(* CODESYS project utilitieslib.library
   Author: Chris van Kooij
   Placeholder: Utilities_Library
   Title: Utilities_Library
   Version: 1.2.0.1
   Description: Utilities library contains all basic utilities needed like system variables messages parameters etc.
   Company: AMKO-Engineering

Project tree, tasks and I/O mapping:
  libraries: Tc2_Standard, * (Beckhoff Automation GmbH); Tc2_System, * (Beckhoff Automation GmbH); Tc2_Utilities, * (Beckhoff Automation GmbH)
  Compare/
    Functions/
      function Between [ST]
      function Between360deg [ST]
  Conversion/
    function DegS_To_Rpm [ST]
    function DegS_To_Rpm_And_MMin [ST]
    function Grey_To_Bin [ST]
    function MMin_To_Rpm_And_DegS [ST]
    function Rpm_To_DegS [ST]
  FaultsAndMessages/
    DataTypes/
      data type E_ComponentTypes
      data type E_FaultTypes
      data type E_Locations
      data type E_MessageNumbers
      data type UDT_Fault
    Functions/
      function block Fb_FaultHandler [ST]: CheckEntryValid, ExecCleanUpArray, ExecResetFaults, ExecSetFaultBit, ExecWriteMessage, CmdAddFault
      function block FB_OperatorMessageDisplay [ST]
    global variables Param_Messages
  General/
    DataTypes/
      data type Udt_TimerBandwith
  GVLs/
    global variables DataManager
    global variables GVL_Message
    global variables GVL_Parameters
    global variables GVL_Safety
    global variables Sys_Variables
  Parameter/
    DataTypes/
      Old/
        data type UDT_Parameter_1
        data type Udt_Parameter_2
        data type Udt_ParameterRetain
      data type E_ParameterNames
      data type Udt_Parameter
      data type Udt_ParameterId
      data type Udt_ParLog
    Functions/
      function block FB_ParameterHandler [ST]: CmdAddParameter, ExecChangeParValues
      function block Fb_ParameterHandlerOld [ST]: Mod_SearchIndex, Mod_WriteTeachValue
      function block Fb_ParLogging [ST]: Init, Mod_CSVFileRead, Mod_CSVFileWrite, Mod_BackupPar, Mod_ChangePar, Mod_ReadAllPar
      global variables Param_Settings
  PathFunctions/
    function F_FBNameFromPath [ST]
  Positions/
    FunctionBlocks/
      function block FB_PositionTrigger [ST]: CalcTriggerCompensation, ExecArmTrigger, ExecTurnoverCheck, CmdArmTrigger, CmdSetTriggerPos
    Functions/
      function F_AccDecDistanceFromTime [ST]
      function F_AccDecDistanceFromVelo [ST]
      function F_PosCheck [ST]
      function F_TopVelocityFromTime [ST]
      function F_TriggerPosOffset [ST]
  System/
    DataTypes/
    Functions/
      DataManagement/
        function block FB_PersistentDataManager [ST]: Write
      function block Fb_SystemVariables [ST]
  Utilities_CD
*)

// FaultsAndMessages/DataTypes/E_ComponentTypes
{attribute 'qualified_only'}
{attribute 'strict'}
{attribute 'to_string'}
TYPE E_ComponentTypes :
(
	// No entry
		NA			:= 0,
	// Actuators 
		Cylinder 	:= 10,
		Axis		:= 11,
	// Buttons 
		EstopButton	:= 20,
		EstopBumper	:= 21,	
		Pushbutton 	:= 22,
		Switch		:= 23,
	// I/O
		SafeIO		:= 30,
		Rio_Box		:= 31,
		Rio_Slot	:= 32,
		Encoder		:= 33,
		DiSensor	:= 34,
	// Drive
		ServoDrive 	:= 40,
	// Operation
		HMI			:= 50,
		RemoteOS	:= 51,
		RemoteDB	:= 52,
	// Assemblies
		Assembly 	:= 60,
		SubAssembly	:= 61,
	// functions
		MainProgram		:= 100,
		StepProgram		:= 101,
		FunctionBlock	:= 102 
)UDINT;
END_TYPE

// FaultsAndMessages/DataTypes/E_FaultTypes
{attribute 'qualified_only'}
{attribute 'strict'}
{attribute 'to_string'}
TYPE E_FaultTypes :
(
	NA	:= 0, // Not applicable
	OM 	:= 1, // Operator message
	MC	:= 2, // Missing condition
	CF	:= 3, // Cycle Fault
	FF	:= 4 // Fatal fault
)UDINT;
END_TYPE

// FaultsAndMessages/DataTypes/E_Locations
{attribute 'qualified_only'}
{attribute 'strict'}
TYPE E_Locations :
(
	MainPLC,
	MainPower_230V, 
	MainPower_24V, 
	MainAirSupply,
	MainScreen,
	MainIO,
	RemoteIO
);
END_TYPE

// FaultsAndMessages/DataTypes/E_MessageNumbers
{attribute 'qualified_only'}
{attribute 'strict'}
TYPE E_MessageNumbers :
(
	// no messages
		NA_NoMessage		:= 0, // no message active
	// System faults
		FF_Unknown 			:= 1, // unknown error occured 
		FF_NoCommunication 	:= 2, // no communication detected
		FF_ComunicationFault:= 3, // Communication error detected (does not match expected com)
		FF_Overload			:= 4, // hardware overload detected
		FF_EncoderFault		:= 5, // encoder signal incorrect or not present
		FF_SlaveFault		:= 6, // slave system is has active fatal fault
		FF_AxisFault		:= 7, // Axis fault feedback
		FF_DriveFault		:= 8, // Axis drive fault
		FF_Collision		:= 9, // Collision detected between 2 or more parts of the machine
	// Hardware faults
		CF_FeedbackFault		:= 100,	// Hardware feedback is does not match expected
		CF_WrongDirection		:= 101, // Hardware moving in incorrect direction
		CF_MoveToFast			:= 102, // Hardware movement completion time is lower then minimum
		CF_MoveToSlow			:= 103, // hardware movement maximum time was exceeded
		CF_WrongPosition		:= 104,	// Hardware is at different position then expected
		CF_Obstruction			:= 105, // Obstruction detected in movement path
	// Missing conditions
		MC_WaitingForproduct	:= 200,	// Waiting for product
		MC_WaitingForOperator	:= 201, // Waiting for operator action
		MC_WaitingForModule		:= 202,	// Waiting for other module
		MC_WaitingForMaster		:= 203, // Waiting Waiting for master
		MC_WaitingForSlave		:= 204, // waiting for slave
		MC_WrongPosition		:= 205, // Action or command not possible in current position
	// Operator messages
		OM_AlmostEmpty			:= 300, // product is almost empty refil is required
		OM_Finished 			:= 301, // product or action is finished
		OM_ready				:= 302, // ready for new task
	// Test Messages
		FF_MessageTest			:= 900, // Fatal fault message test
		CF_MessageTest			:= 901, // Cycle fault message test
		MC_MessageTest			:= 902, // Missing condition message test
		OM_MessageTest			:= 903	// Operator message test
)UDINT;
END_TYPE

// FaultsAndMessages/DataTypes/UDT_Fault
TYPE UDT_Fault :
STRUCT
	// active 
		Active 			: BOOL 				:= FALSE;
	// Message type
 		FaultType 		: E_FaultTypes 		:= E_FaultTypes.NA; // Type of message
	// Message Id number used for translation
		MessageNumber 	: UDINT				:= 0; // message number
		LocationNumber	: UDINT 			:= 0; // message number array ([1]= System, [2]= Module,[3]= sub module, [4]= Component)
	// Message discription
		Discription 	: STRING 			:= ''; // Message text discription in english (service personel only)
	// Location
		LocationName	: STRING			:= ''; // Location discription name
		ComponentType 	: E_ComponentTypes 	:= E_ComponentTypes.NA; // Part type discription
	// Time stamp
		StartTime		: DATE_AND_TIME 	:= DT#2020-1-1-00:00:00 ; // Time and date of message occurence
		EndTime			: DATE_AND_TIME		:= DT#2020-1-1-00:00:00 ; // Time and date of message end
	// Module number
		nModuleID		: UDINT 			; // module reference number used for fault, enable, reset, and safety functions (default := 1, 0 = main system)
	// CompleteFaultnumber for visualization
		FullFaultId		: STRING 			:= 'NA.0.0.0'; // Full fault id for use in HMI is writen by fault function [fault type, message#, location#,ComponentType]
END_STRUCT
END_TYPE

// General/DataTypes/Udt_TimerBandwith
TYPE Udt_TimerBandwith :
STRUCT
	Minimal	:LREAL;// Timer values, Minimum time
	Nominal	:LREAL;// timer values, nominal time
	Maximum	:LREAL;// Timer values, Maximum time
END_STRUCT
END_TYPE

// Parameter/DataTypes/Old/UDT_Parameter_1
TYPE UDT_Parameter_1 EXTENDS Udt_ParameterRetain:
STRUCT
	Name		: STRING	; // Parameter data, Parameter name
	Number		: INT		; // Parameter data, Parameter number
	Par_TYPE	: STRING	; // Parameter data, Type of parameter [Mpar, Cpar, Opar, Ppar]
	Discription	: STRING	; // Parameter data, Parmater discription
	Factory		: LREAL		; // Parameter data, Factory standard value
	Maximum		: LREAL		; // Parameter data, Maximum parameter value
	Minimum		: LREAL		; // Parameter data, Minimum parameter value
	Unit		: STRING	; // Parameter data, Unit of measurement
END_STRUCT
END_TYPE

// Parameter/DataTypes/Old/Udt_Parameter_2
TYPE Udt_Parameter_2 :
STRUCT
	bActive		: BOOL 	; // True if parameter is active in machine 
	IndexNumber	: UDINT	; // [Column 0] Array row index number  
	Number		: INT	; // [Column 1]Parameter data, parameter number
	Name		: STRING; // [Column 2]Parameter data, Parameter name
	Par_Type	: STRING; // [Column 3]Parameter data, Type of parameter [Mpar, Cpar, Opar, Ppar]
	Discription	: STRING; // [Column 4]Parameter data, Parmater discription
	Factory		: LREAL	; // [Column 5]Parameter data, Factory standard value
	Maximum		: LREAL	; // [Column 6]Parameter data, Maximum parameter value
	Minimum		: LREAL	; // [Column 7]Parameter data, Minimum parameter value
	Unit		: STRING; // [Column 8]Parameter data, Unit of measurement
	Value		: LREAL	; // [Column 9]Parameter data, Current (active) parameter value
	Saved		: LREAL	; // [Column 10]Parameter data, Saved value or standard setpoint
	bCmdTeach	: BOOL	; // Teach command for devices 
	bCmdSave	: BOOL 	; // Command to parameter handler to save the parameter
//	LastChange	: DT	; // [Column 11]Parameter data, Date of last change
END_STRUCT
END_TYPE

// Parameter/DataTypes/Old/Udt_ParameterRetain
TYPE Udt_ParameterRetain :
STRUCT
	PrepValue	: LREAL		; // Parameter data, prepared value
	Value		: LREAL		; // Parameter data, Current (active) parameter value
	Saved		: LREAL		; // Parameter data, Saved value or standard setpoint
	LastChange	: DT		; // Parameter data, Date of last change
END_STRUCT
END_TYPE

// Parameter/DataTypes/E_ParameterNames
{attribute 'qualified_only'}
{attribute 'strict'}
TYPE E_ParameterNames :
(
	Mpar_StitchLengthLong 			,
	MPar_StitchLengthShort 			,
	MPar_MaxSpeed 					,
	Mpar_MinSpeed 					,
	Mpar_ManualMaxSpeed 			,
	Mpar_BacktackSpeed 				,
	Mpar_SlowEndSpeed 				,
	Mpar_HomingSpeed 				,
	Mpar_CuttingSpeed 				,
	Mpar_MaxAcceleration 			,
	Mpar_MaxDeceleration 			,
	Mpar_Jerk 						,
	Mpar_BacktackAcceleration 		,
	Mpar_BacktackDeceleration 		,
	Mpar_TransferAcceleration 		,
	Mpar_TransferDeceleration 		,
	Mpar_CylinderTimeoutMargin		,
	Cpar_NeedleSensorPos 			,
	Cpar_NeedlePosUp 				,
	Cpar_NeedlePosInMaterial 		,
	Cpar_NeedleposDown 				,
	Cpar_NeedlePosStartCut 			,
	Cpar_NeedlePosStopCut 			,
	Cpar_NeedlePosEndCut 			,
	Cpar_NeedlePosRelTensCut 		,
	Cpar_NeedlePosHoldThread 		,
	Cpar_NeedlePosStartRelTension 	,
	Cpar_NeedlePosStopRelTension 	,
	Cpar_NeedlePosChangeDirUp 		,
	Cpar_NeedlePosClearStart 		,
	Cpar_NeedlePosClearEnd 			,
	Cpar_NeedlePosRef 				,
	Cpar_NeedlePosPause 			,
	Cpar_SensorPreEdgeDetDistance 	,
	Cpar_sensorEdgeDetDistance 		,
	Opar_NeedleSensorPos 			,
	Opar_NeedlePosUp 				,
	Opar_NeedlePosInMaterial 		,
	Opar_NeedleposDown 				,
	Opar_NeedlePosStartCut 			,
	Opar_NeedlePosStopCut 			,
	Opar_NeedlePosEndCut 			,
	Opar_NeedlePosRelTensCut 		,
	Opar_NeedlePosHoldThread 		,
	Opar_NeedlePosStartRelTension 	,
	Opar_NeedlePosStopRelTension 	,
	Opar_NeedlePosChangeDir 		,
	Opar_NeedlePosClearStart 		,
	Opar_NeedlePosClearEnd 			,
	Opar_NeedlePosPause 			,
	Ppar_BacktackStitchStartFwd 	,
	Ppar_BacktackStitchStartRev 	,
	Ppar_BacktackStitchEndFwd 		,
	Ppar_BacktackStitchEndRev 		,
	Ppar_AutomaticSpeed 			,
	Ppar_StitchStretch 				,
	Ppar_ThreadLengthAdition 		,
	Ppar_ThreadBreakDelay 			,
	Mpar_MaxVelocity 				,
	Mpar_MinVelocity 				,
	Mpar_ManualMaxVelocity 			,
	Mpar_MLTMaxAcceleration 		,
	Mpar_MLTMaxDeceleration 		,
	Mpar_TraverseLength 			,
	Mpar_CylTimeOutMargine 			,
	Mpar_HomingVelocity 			,
	Mpar_SewingcartLength 			,
	Mpar_ClampCartLength 			,
	Mpar_MaxClampCartVelocity 		,
	Mpar_TraverseReturnVelocity 	,
	Mpar_ToStartvelocity 			,
	Mpar_InspectionDistance 		,
	Cpar_PosHoming 					,
	Cpar_PosSuportCyl_1 			,
	Cpar_PosSuportCyl_2 			,
	Cpar_PosSuportCyl_3 			,
	Cpar_PosService 				,
	Cpar_PosBobinChange 			,
	Cpar_PosEnd 					,
	Cpar_TimeBaseClampsClose 		,
	Cpar_TimeBaseClampsRel 			,
	Cpar_TimeCartClampsClose 		,
	Cpar_TimeCartClampsRel 			,
	Cpar_TimeCartBrakeApply 		,
	Cpar_TimeCartBrakeRel 			,
	Cpar_TimeSupportExp_1 			,
	Cpar_TimeSupportRet_1 			,
	Cpar_TimeSupportExp_2 			,
	Cpar_TimeSupportRet_2 			,
	Cpar_TimeSupportExp_3 			,
	Cpar_TimeSupportRet_3 			,
	Cpar_TimeBobinPlateClose 		,
	Cpar_TimeBobinPlateOpen 		,
	Cpar_PosFlagSewingcart 			,
	Cpar_PosSensorClampCart 		,
	Cpar_SupportCylWidth 			,
	Cpar_ClampCartFlagWidth 		,
	Cpar_PosMaterialStart 			,
	Opar_HomePosition 				,
	Opar_PosSuportCyl_1 			,
	Opar_PosSuportCyl_2 			,
	Opar_PosSuportCyl_3 			,
	Opar_PosService 				,
	Opar_PosBobinChange 			,
	Opar_PosEnd 					,
	Opar_PosMatStart 				,
	Ppar_ProductLenght 				,
	Ppar_ProductStretch 			,
	Ppar_StartStretchFactor 		,
	Ppar_StartStretchLength 		,
	Ppar_ReverseStretch 			,
	Ppar_MatBlowDistance 			 
)UDINT;
END_TYPE

// Parameter/DataTypes/Udt_Parameter
TYPE Udt_Parameter :
STRUCT
	nNumber		: INT	 	:= 0				; // [Column 1]Parameter data, parameter number
	sName		: STRING	:= 'No parameter' 	; // [Column 2]Parameter data, Parameter name
	sType		: STRING	:= 'PPar'			; // [Column 3]Parameter data, Type of parameter [Mpar, Cpar, Opar, Ppar]
	sDiscription: STRING	:= 'No parameter selcted'; // [Column 4]Parameter data, Parmater discription
	fFactory	: LREAL		:= 0				; // [Column 5]Parameter data, Factory standard value
	fMaximum	: LREAL		:= 0				; // [Column 6]Parameter data, Maximum parameter value
	fMinimum	: LREAL		:= 0				; // [Column 7]Parameter data, Minimum parameter value
	sUnit		: STRING	:= 'na'				; // [Column 8]Parameter data, Unit of measurement
	fValue		: LREAL		:= 0				; // [Column 9]Parameter data, Current (active) parameter value
	fSaved		: LREAL		:= 0				; // Parameter data, Saved value or standard setpoint
	fPrepared	: LREAL 	:= 0				; // Parameter data, Prepared value from teach function 
	bCmdTeach	: BOOL		:= FALSE			; // Teach command for devices 
END_STRUCT
END_TYPE

// Parameter/DataTypes/Udt_ParameterId
TYPE Udt_ParameterId :
STRUCT
	nNumber		: INT 		:= 0 	; // parameter number
	sName		: STRING 	:= 'NA' ; // parameter name
	sType		: STRING 	:= 'Ppar'	; // parameter type 
	pParameter	: POINTER TO Udt_Parameter ; // pointer to parameter
END_STRUCT
END_TYPE

// Parameter/DataTypes/Udt_ParLog
TYPE Udt_ParLog :
STRUCT
	ParList		: ARRAY [0..Param_Settings.MAX_PARAMETERS] OF Udt_Parameter_2 ; // active parameter list
END_STRUCT
END_TYPE

// FaultsAndMessages/Param_Messages
{attribute 'qualified_only'}
VAR_GLOBAL CONSTANT
	nMAX_MESSAGES_SHOWN 	: UDINT := 10 	;
	nMAX_MESSAGE_HISTORY	: UDINT := 1000 ;
	nMAX_CSV_FIELD_LENGTH	: UDINT := 100	;
	tMESSAGE_TIMEOUT		: TIME 	:= T#5S ;
	sLOGFILE_PATH			: STRING:= 'C:\FaultLogs\'	;
	sLOGFILE_NAME			: STRING:= 'Faultlog' 		; // Message log destination file
	nMESSAGE_COLUMNS		: UDINT := 8 ;
	
END_VAR

// GVLs/DataManager
{attribute 'qualified_only'}
VAR_GLOBAL
	FbPersistentManager : FB_PersistentDataManager ;
END_VAR

// GVLs/GVL_Message
{attribute 'qualified_only'}
VAR_GLOBAL
	bResetFaults		: BOOL 	:= FALSE	; // Reset system faults 
	bCmdSnoozeMessage	: BOOL 	:= FALSE	; // Snooze message display
	bDisplayFaults		: BOOL := FALSE 	; // Display fault message popup on screen (when MC, CF of FF are active)
	arActiveFaults 		: ARRAY [0..Param_Messages.nMAX_MESSAGES_SHOWN] OF UDT_Fault ; // Active faults overview for showing in HMI
END_VAR
VAR_GLOBAL CONSTANT 
	tMESSAGESNOOZEDURATION	: TIME 	:= T#5s ; // duration of message snooze after button press 
END_VAR

// GVLs/GVL_Parameters
{attribute 'qualified_only'}
VAR_GLOBAL
	fbParameterHandler	: FB_ParameterHandler ; // Default parameter handler for visualisation and file handling
END_VAR

// GVLs/GVL_Safety
{attribute 'qualified_only'}
VAR_GLOBAL
	// ===== system Safety inputs =====
		SafeCom_SystemSafe		AT %I* : BOOL ; // System safety communication safety system is running
		SafeCom_EstopOk			AT %I* : BOOL ; // System safety communication emergency stop active
		SafeCom_BumpersOk		AT %I* : BOOL ; // System safety communication safety zone tripped
		SafeCom_ComError		AT %I* : BOOL ; // System safety communication Common error active in safety program
		
		SafeCom_EstopReset		AT %Q* : BOOL ; // System Safety Communication Safety Reset 
		SafeCom_RunSafety		AT %Q* : BOOL ; // System Safety Communication Run safety program
		SafeCom_AcnSafeError	AT %Q* : BOOL ; // System Safety Communication acknowlidge safety error		 
		SafeCom_ResetActive		AT %Q* : BOOL ; // System safety communication reset active
		Safecom_BumperReset		AT %Q* : BOOL ; // System safety communication reset safety bumpers 
		SafeCom_EnableOff		AT %Q* : BOOL ; // System Safety communication motor enable signals are off
		
		SafeOp_AirPressureOk	AT %I* : BOOL ; // system safety condition monitorring air pressure ok
		SafeOp_PowerSupplyOk	AT %I* : BOOL ; // System power supply is ok
END_VAR

// GVLs/Sys_Variables
(* System variables *)
{attribute 'qualified_only'}
VAR_GLOBAL
// SystemFuntion
	fbSystemVariables : Fb_SystemVariables ;
	AlwaysOn		:BOOL 			;// System variable, Always on bit
	AlwaysOff		:BOOL 			;// System variable, Always off bit
	BlinkFast		:BOOL 			;// System variable, Blink fast bit 1sec 
	BlinkSlow		:BOOL 			;// System variable, Blink slow bit 2 sec
	Pulse1Sec		:BOOL 			;// System variable, Pulse 1 cycle every second
	SystemTime		:DT				; // System variable, Windows system time
	TimeZoneId		:E_TimeZoneID 	; // System variable, time zone Id 
	HeartBeat		:BOOL 			;// System Variable, Main system heartbeat 0.5 sec on 0.5 sec off
END_VAR

// Parameter/Functions/Param_Settings
{attribute 'qualified_only'}
VAR_GLOBAL CONSTANT
	MAX_PARAMETERS 			: UDINT := 1000	;
	PAR_COLUMNS 			: UDINT := 11	;
	MAX_CSV_FIELD_LENGTH	: UDINT := 100	;
	sPARLIST_FILE			: T_MaxString 		:= 'C:\Users\chris\Documents\TestCsvList.csv';(* CSV destination file path and name *)
	sPARLOG_FILE			: T_MaxString 		:= 'C:\Users\chris\Documents\TestCsvLog.csv';(* CSV destination file path and name *)
	sNetId					: T_AmsNetID		:= '' ;
END_VAR

// Compare/Functions/Between
FUNCTION Between : BOOL // Returns true if value is >= the lower and <= the upper threshold
VAR_INPUT
	Lower	: LREAL	; // lower threshold value [LREAL]
	Value	: LREAL	; // test value [LREAL]
	Upper	: LREAL	; // Upper threshold value [LREAL]
END_VAR
VAR
END_VAR

// Check if value is between lower and upper threshold
Between := (Value >= Lower) AND (Value <= Upper);

END_FUNCTION

// Compare/Functions/Between360deg
FUNCTION Between360deg : BOOL // Returns true if value is >= the lower and <= the upper threshold, if lower > upper then upper := Upper +360 deg
VAR_INPUT
	Lower	: LREAL	; // lower threshold value [LREAL]
	Value	: LREAL	; // test value [LREAL]
	Upper	: LREAL	; // Upper threshold value [LREAL]
END_VAR
VAR
END_VAR

IF Lower > Upper THEN  
	Between360deg S= Between( Lower, Value, 360);
	Between360deg S= Between( 0, Value, Upper)	;
ELSE 
	Between360deg S= Between( Lower, Value, Upper)	;
END_IF

END_FUNCTION

// Conversion/DegS_To_Rpm
(* convert degrees per second to rotations per minute *)
FUNCTION DegS_To_Rpm : LREAL
VAR_INPUT
	DegS : LREAL ; // Input degrees per second as long real
END_VAR

// ===== convert degrees per second to Rpm =====
	DegS_To_Rpm := (DegS/360)*60 ;

END_FUNCTION

// Conversion/DegS_To_Rpm_And_MMin
FUNCTION DegS_To_Rpm_And_MMin : BOOL
VAR_INPUT
	DegPerSecond : LREAL ; // Input degrees per second
	StitchLength : LREAL ; // Input stitch length
END_VAR
VAR_OUTPUT
	RevPerMinute	: LREAL ; // Output revolutions per minute
	MetersPerMinute	: LREAL ; // Output meters per minute
END_VAR
VAR
END_VAR

// ===== convert degrees per second to Rpm =====
	RevPerMinute := (DegPerSecond/360)*60 ;
// ===== Convert RPM to MMin =====
	MetersPerMinute := RevPerMinute * StitchLength / 1000 ;

END_FUNCTION

// Conversion/Grey_To_Bin
FUNCTION Grey_To_Bin : INT // convert 4 bit grey code into 8 bit binary code
VAR_INPUT
	GreyBit0 : BOOL := FALSE ;
	GreyBit1 : BOOL := FALSE ;
	GreyBit2 : BOOL := FALSE ;
	GreyBit3 : BOOL := FALSE ;
END_VAR
VAR
	TempInt : INT ; // temporary 
END_VAR

// convert grey code into binary
TempInt.3 	:= GreyBit3 ;
TempInt.2	:= GreyBit3 	XOR GreyBit2 ;
TempInt.1	:= TempInt.2	XOR GreyBit1 ;
TempInt.0	:= TempInt.1	XOR GreyBit0 ;

Grey_To_Bin := TempInt ;

END_FUNCTION

// Conversion/MMin_To_Rpm_And_DegS
(* Convert meters per minute to degrees per second *)
FUNCTION MMin_To_Rpm_And_DegS : BOOL
VAR_INPUT
	MeterPerMinute 	: LREAL ; // Input meters per minute
	StitchLength	: LREAL ; // Input Stitch length
END_VAR
VAR_OUTPUT
	RevPerMinute	: LREAL ; // Output revolutions per minute
	DegPerSecond	: LREAL ; // Output degrees per second
END_VAR
VAR
	MmMin 	: LREAL ; // Millimeters per minute
	RevSec 	: LREAL ; // Millimeters per second
END_VAR

// ===== convert MMin to RPM =====
	RevPerMinute := (MeterPerMinute * 1000) / StitchLength ;
//===== Convert RPM to DegS =====
	DegPerSecond := (RevPerMinute/60)*360 ;

END_FUNCTION

// Conversion/Rpm_To_DegS
(* convert rotations per minute to degrees per second *)
FUNCTION Rpm_To_DegS : LREAL 
VAR_INPUT
	Rpm : LREAL ; // input revolutions per minute
END_VAR

// ===== convert RPM to DegS ====
	Rpm_To_DegS := (Rpm/60)*360 ;

END_FUNCTION

// FaultsAndMessages/Functions/Fb_FaultHandler
FUNCTION_BLOCK Fb_FaultHandler
VAR_INPUT
	bReset 				: BOOL 	:= FALSE	; // reference to fault reset bit
END_VAR
VAR_OUTPUT
	arActiveFaults 	: ARRAY [0..Param_Messages.nMAX_MESSAGES_SHOWN] OF UDT_Fault  ; // reference to active fault array
	nActiveFaults	: UDINT 			; // reference to active fault counter
	bActOM 			: BOOL := FALSE ;
	bActMC 			: BOOL := FALSE ;
	bActCF 			: BOOL := FALSE ;
	bActFF 			: BOOL := FALSE ;
END_VAR
VAR
	// functional variables
	i 					: UDINT ;
	// fault data
	stFaultUdt 			: UDT_Fault ;
	bTimedOut 			: BOOL ; // Message has timed out
	// Message logging
	dToday				: DATE ; 
	nWriteStep			: UDINT := 0 ;
	bWriteError			: BOOL 	; // write to file error occured
	nWriteErroId		: UDINT ; // write error id
	// Write variables
	sActFileName		: STRING ;
	hFile				: UINT	:= 0;(* File handle of the source file *)
	sMessageString		: ARRAY [0..Param_Messages.nMESSAGE_COLUMNS] OF STRING (Param_Settings.MAX_CSV_FIELD_LENGTH); (* temporary parameter buffer to string*)
	sCSVLine			: T_MaxString := '';(* Single CSV text line (row, record), we are using string as record buffer (your are able to see created fields) *)
	sCSVField			: T_MaxString := '';(* Single CSV field value (column, record field) *)

	// Log to file functions
	fbFileOpen		: FB_FileOpen	;(* Opens file *)
	fbFileClose		: FB_FileClose	;(* Closes file *)
	fbFileGets		: FB_FileGets	;(* Reads one record (line) *)
	fbFilePuts		: FB_FilePuts	;(* Writes one record (line) *)
	fbReader		: FB_CSVMemBufferReader;(* Helper function block used to parse CSV data bytes (single record line) *)
	fbWriter		: FB_CSVMemBufferWriter;(* Helper function block used to create CSV data bytes (single record line) *)
END_VAR
VAR PERSISTENT
	dLastFileDate : DATE ;
END_VAR
VAR CONSTANT
	stEmptyMessageUdt : UDT_Fault := (	Active 			:= FALSE,
										FaultType 		:= E_FaultTypes.NA,
										MessageNumber	:= 0,
										LocationNumber	:= 0,
										Discription 	:= '',
										LocationName	:= '',
										ComponentType	:= E_ComponentTypes.NA,
										StartTime		:= DT#2020-1-1-00:00:00,
										EndTime			:= DT#2020-1-1-00:00:00,
										FullFaultId		:= '0'	)  ;
END_VAR

// Check for active faults in list
ExecSetFaultBit(); 
// Check for reset is active 
ExecResetFaults();

METHOD PRIVATE CheckEntryValid : BOOL
VAR
	// functional variables
	i 	: UDINT ;
END_VAR
// ======= check if new entry is valid and not already active ======
CheckEntryValid S= TRUE ;
FOR i := 0 TO nActiveFaults DO
	IF arActiveFaults[i].MessageNumber = stFaultUdt.MessageNumber THEN 
		CheckEntryValid 			:= FALSE ; 
		arActiveFaults[i].Active 	:= TRUE ; 
	END_IF
END_FOR
END_METHOD

METHOD PRIVATE ExecCleanUpArray : BOOL
VAR
	// functional variables
	i 					: UDINT ;
END_VAR
// Clean up array by removing blanc spaces 
REPEAT
	IF arActiveFaults[i].FaultType = 0 THEN 
		arActiveFaults[i] 	:= arActiveFaults[i+1];
		arActiveFaults[i+1] := stEmptyMessageUdt;
	END_IF
	i := i +1 ;
UNTIL 
	i = Param_Messages.nMAX_MESSAGES_SHOWN   
END_REPEAT
END_METHOD

METHOD PRIVATE ExecResetFaults : BOOL
VAR
	nResetPoint : UDINT := 0 ; // point of reset for active fault array (skips fault if .active bit is true)
	// functional variables
	i 					: UDINT ;
END_VAR
IF NOT bReset THEN 
	RETURN;
END_IF

FOR i := 0 TO Param_Messages.nMAX_MESSAGES_SHOWN DO
	IF arActiveFaults[i].Active THEN
		CONTINUE;
	ELSE
		arActiveFaults[i] := stEmptyMessageUdt; 
	END_IF
END_FOR

ExecCleanUpArray();

bActOM 			:= FALSE;
bActMC 			:= FALSE;
bActCF 			:= FALSE;
bActFF 			:= FALSE;

ExecResetFaults := TRUE ;
END_METHOD

METHOD PRIVATE ExecSetFaultBit : BOOL
bActOM 	:= FALSE;
bActMC	:= FALSE;
bActCF 	:= FALSE;
bActFF 	:= FALSE;

FOR i := 0 TO nActiveFaults DO
	// read message type 
	CASE arActiveFaults[i].FaultType OF
		E_FaultTypes.OM : 
			IF arActiveFaults[i].Active THEN 
				bActOM 		S= TRUE ;
			ELSE 
				bTimedOut 	S= TRUE ;
			END_IF 
		E_FaultTypes.MC :
			IF arActiveFaults[i].Active THEN 
				bActMC 		S= TRUE ;
			ELSE 
				bTimedOut 	S= TRUE ;
			END_IF 
		E_FaultTypes.CF:
			bActCF 		S= TRUE ;
		E_FaultTypes.FF:
			bActFF 		S= TRUE ;
		ELSE
			bTimedOut := FALSE ;
	END_CASE

	IF bTimedOut THEN 
		arActiveFaults[i] := stEmptyMessageUdt;				
		bTimedOut := FALSE ;
	END_IF
	// Reset active bit when timed out, if fault is still active it will be set to true again.
	arActiveFaults[i].Active R= (arActiveFaults[i].StartTime + Param_Messages.tMESSAGE_TIMEOUT) < Sys_Variables.SystemTime;
END_FOR

// clean up the fault array
ExecCleanUpArray();
END_METHOD

ACTION ExecWriteMessage:
// Set message start time 
stFaultUdt.StartTime := Sys_Variables.SystemTime ;
// Fill Full Fault Id
stFaultUdt.FullFaultId := TO_STRING(stFaultUdt.FaultType);
stFaultUdt.FullFaultId := CONCAT(stFaultUdt.FullFaultId,'.');
stFaultUdt.FullFaultId := CONCAT(stFaultUdt.FullFaultId,UDINT_TO_STRING(stFaultUdt.MessageNumber));
stFaultUdt.FullFaultId := CONCAT(stFaultUdt.FullFaultId,'.');
stFaultUdt.FullFaultId := CONCAT(stFaultUdt.FullFaultId,UDINT_TO_STRING(stFaultUdt.LocationNumber));
stFaultUdt.FullFaultId := CONCAT(stFaultUdt.FullFaultId,'.');
stFaultUdt.FullFaultId := CONCAT(stFaultUdt.FullFaultId,UDINT_TO_STRING(stFaultUdt.ComponentType));
// send message to higher level 
arActiveFaults[nActiveFaults] := stFaultUdt		;
// Set pointer to next fault
IF nActiveFaults < Param_Messages.nMAX_MESSAGES_SHOWN THEN 
	nActiveFaults := nActiveFaults + 1 	;
ELSE
	nActiveFaults := 0 ;
END_IF
END_ACTION

METHOD PUBLIC CmdAddFault : BOOL
VAR_IN_OUT
	stFault : UDT_Fault ; // actuive fault structure input
END_VAR

// coppy fault to internal fault udt
IF stFault.FaultType <> E_FaultTypes.NA THEN 
	THIS^.stFaultUdt	:= stFault ;
	stFault 			:= stEmptyMessageUdt ;
	stFaultUdt.Active	:= TRUE ;
	// Process fault data
	IF CheckEntryValid() THEN
		ExecWriteMessage();
	END_IF
END_IF
END_METHOD

END_FUNCTION_BLOCK

// FaultsAndMessages/Functions/FB_OperatorMessageDisplay
FUNCTION_BLOCK FB_OperatorMessageDisplay // function compares messages and shows latest message on screen for a set period of time
VAR_INPUT
	bEnable 	: BOOL 	:= TRUE ; // enable messages
	tDisplayTime: TIME	:= Param_Messages.tMESSAGE_TIMEOUT ; // Time before message relevance is checked (default = Param_Messages.tMESSAGE_TIMEOUT)
END_VAR
VAR_IN_OUT
	sMessage 	: STRING ; // Operator message (default = GVL_Message.sOPeratorMessage)
END_VAR
VAR_OUTPUT
	sOutMessage : STRING ; // message output to screen
END_VAR
VAR
	sOldMessage 	: STRING := ''; // old message as displayed 
	tonDisplayTimer	: TON ; // Display timer
END_VAR

// Run timers
tonDisplayTimer(PT := tDisplayTime);

// compare old message with new message 
IF sMessage = sOldMessage THEN 
	tonDisplayTimer.IN := TRUE ;
	IF tonDisplayTimer.Q = TRUE THEN 
		sMessage := '';
	END_IF
ELSE 
	tonDisplayTimer.IN 	:= FALSE 	;
	sOldMessage 		:= sMessage ; 
END_IF

// write message to display
sOutMessage := sMessage ;

END_FUNCTION_BLOCK

// Parameter/Functions/FB_ParameterHandler
FUNCTION_BLOCK PUBLIC FB_ParameterHandler
VAR_INPUT
END_VAR
VAR_OUTPUT
	arParameters		: ARRAY [0..Param_Settings.MAX_PARAMETERS] OF Udt_ParameterId := [stDummyParId]; 
END_VAR
VAR
	nLookupIndex		: UDINT := 0;
	nNumberOfParameters : UDINT := 0;
	// parameter change commands
	bCmdLoadfactory		: BOOL 	:= FALSE; // Load factory value into prepared value 
	bCmdLoadFromPrevious: BOOL 	:= FALSE; // Load from saved previous value into prepared value
	bCmdTeach			: BOOL 	:= FALSE; // Start teaching function for selected parameter
	bCmdAcceptTeach		: BOOL 	:= TRUE ; // Accept the teach value
	// Dummy parameter when no parameters are added yet
	stDummyParId		: Udt_ParameterId ;
	// Memory 
	fValueOld			: LREAL	:= 0 ; // previous value
END_VAR

// call parameter change function 
ExecChangeParValues();

METHOD PUBLIC CmdAddParameter : BOOL
VAR_INPUT
	refParameter : REFERENCE TO Udt_Parameter ; // reference to parameter 
END_VAR
VAR
	i 			: UDINT ;
	j			: UDINT ;
	stTempPar	: Udt_ParameterId ;
	bParFound	: BOOL 	:= FALSE ;
END_VAR
// check if parameter is already added
FOR i := 0 TO Param_Settings.MAX_PARAMETERS DO
	IF arParameters[i].pParameter = 0 THEN 
		nNumberOfParameters := i;
		EXIT ;
	ELSIF arParameters[i].nNumber = refParameter.nNumber THEN
 		RETURN ;
	END_IF
END_FOR
	
// Add parameter to array if not already added
arParameters[nNumberOfParameters].nNumber		:= refParameter.nNumber 	;
arParameters[nNumberOfParameters].sName			:= refParameter.sName	;
arParameters[nNumberOfParameters].sType			:= refParameter.sType	;
arParameters[nNumberOfParameters].pParameter 	:= ADR(refParameter)	;

IF nNumberOfParameters > 1 THEN 
	// (re)sort parameter list
	FOR i := 0 TO nNumberOfParameters BY 1 DO
		FOR j := 0 TO nNumberOfParameters -1 BY 1 DO
			IF (arParameters[j].nNumber > arParameters[j+1].nNumber)THEN
				stTempPar 			:= arParameters[j+1];
				arParameters[j+1]	:= arParameters[j];
				arParameters[j]		:= stTempPar ;
			END_IF
		END_FOR
	END_FOR	
END_IF

// set feedback
CmdAddParameter S= arParameters[nNumberOfParameters].pParameter > 0 ;
END_METHOD

METHOD ExecChangeParValues : BOOL
VAR
END_VAR
IF arParameters[nLookupIndex].pParameter <> 0 THEN 
	;
ELSE
	RETURN; 
END_IF

// Load values from default or saved
IF bCmdLoadfactory THEN 
	arParameters[nLookupIndex].pParameter^.fValue := arParameters[nLookupIndex].pParameter^.fValue ;
ELSIF bCmdLoadFromPrevious THEN
	arParameters[nLookupIndex].pParameter^.fValue := arParameters[nLookupIndex].pParameter^.fSaved ;
ELSIF bCmdAcceptTeach THEN 
	arParameters[nLookupIndex].pParameter^.fValue := arParameters[nLookupIndex].pParameter^.fPrepared ;
END_IF

	// Save current actual value for later restore
IF arParameters[nLookupIndex].pParameter^.fValue <> fValueOld THEN
	arParameters[nLookupIndex].pParameter^.fSaved := fValueOld ;
	fValueOld := arParameters[nLookupIndex].pParameter^.fValue ;
END_IF
END_METHOD

END_FUNCTION_BLOCK

// Parameter/Functions/Fb_ParameterHandlerOld
FUNCTION_BLOCK PUBLIC Fb_ParameterHandlerOld EXTENDS Fb_ParLogging 
VAR_INPUT
	bCmdScrollUp	: BOOL 	:= FALSE; // command to scroll to next parameter
	bCmdScrollDown	: BOOL 	:= FALSE; // command to scroll to previous parameter
	bCmdAccept		: BOOL 	:= FALSE; // Accept parameter and coppy prev value into value
	bCmdSave		: BOOL 	:= FALSE; // save active value into memory 
	bCmdLoad		: BOOL 	:= FALSE; // Load value from memory into prepared value
	bCmdRestore		: BOOL 	:= FALSE; // load Factory value into prepared value
	bCmdRestoreAll	: BOOL 	:= FALSE; // Restore all values to factory default
	bCmdSaveToFile 	: BOOL 	:= FALSE; // Save all parameters to .csv file
END_VAR
VAR_IN_OUT
	PrepValue	: LREAL	:= 0 ; // Parameter data, prepared value
END_VAR
VAR_OUTPUT
	stParToHMI	: Udt_Parameter_2 ; // Parameter that can be shown on HMI 
	bReady		: BOOL 	; // function is ready for new command
	bBussy		: BOOL 	; // Function is bussy
	nProgress	: UDINT ; // Progress for visu [%] 
	bDone		: BOOL 	; // Function is done 
END_VAR
VAR
	CmdIndex	: UDINT ; // Index number of parameter
	
	// ====== functions ======
		rtCmdScrollUp	: R_TRIG; // command to scroll to next parameter
		rtCmdScrollDown	: R_TRIG; // command to scroll to previous parameter
		rtCmdAccept		: R_TRIG; // Accept parameter and coppy prev value into value
		rtCmdSave		: R_TRIG; // save active value into memory 
		rtCmdLoad		: R_TRIG; // Load value from memory into prepared value
		rtCmdRestore	: R_TRIG; // load Factory value into prepared value
		rtCmdSaveToFile : R_TRIG; // Save all parameters to .csv file
		rtCmdTeach		: R_TRIG; // Triger 

	// ====== Teach functions =======
		bCmdTeach		: BOOL 	:= FALSE; // Place teach value in parameter

END_VAR

SUPER^();

// ====== Create rising edges ======
	rtCmdScrollUp	(CLK := bCmdScrollup);
	rtCmdScrollDown	(CLK := bCmdScrollDown);
	rtCmdAccept		(CLK := bCmdAccept);
	rtCmdSave		(CLK := bCmdSave);
	rtCmdLoad		(CLK := bCmdLoad);
	rtCmdRestore	(CLK := bCmdRestore);
	rtCmdSaveToFile	(CLK := bCmdSaveToFile);
	rtCmdTeach		(CLK := bCmdTeach);
	
// call search index 
	IF NOT bCmdTeach THEN 
		Mod_SearchIndex();
	END_IF
	
// ====== Always check if prepared value is within min max range ======
	PrepValue := LIMIT (stParLog.ParList[CmdIndex].Minimum, PrepValue, stParLog.ParList[CmdIndex].Maximum);

// ====== process parameter Prep value ======
	IF rtCmdRestore.Q THEN 
		PrepValue := stParLog.ParList[CmdIndex].Factory ;
	ELSIF rtCmdLoad.Q THEN 
		PrepValue := stParLog.ParList[CmdIndex].Saved	;
	ELSIF rtCmdSave.Q THEN 
		stParLog.ParList[CmdIndex].Saved := stParLog.ParList[CmdIndex].Value ; 
	ELSIF rtCmdAccept.Q THEN 
		stParLog.ParList[CmdIndex].Value := PrepValue ;
	ELSIF rtCmdTeach.Q THEN 
		stParLog.ParList[CmdIndex].Value := PrepValue ;
		bCmdTeach 		:= FALSE ;
		bCmdWriteAllPar := TRUE ;
	END_IF		

// ======= check for missing values and restore to factory ======
	IF stParLog.ParList[CmdIndex].Value = 0 AND stParLog.ParList[CmdIndex].Minimum >0 THEN 
		stParLog.ParList[CmdIndex].Value := PrepValue := stParLog.ParList[CmdIndex].Factory ;
	END_IF

// ======= Restore all values to factory default =======
	IF bCmdRestoreAll THEN 
		FOR CmdIndex := 0 TO Param_Settings.MAX_PARAMETERS BY 1 DO
			IF stParLog.ParList[CmdIndex].bActive THEN  
				stParLog.ParList[CmdIndex].Value := PrepValue := stParLog.ParList[CmdIndex].Factory ;
			END_IF
		END_FOR
	END_IF
	
// ======= save parameters to file =======
	IF rtCmdSaveToFile.Q THEN
		bCmdWriteAllPar := TRUE ;
	END_IF
		 
// ======= set feedback to HMI =====
	stParToHMI :=  stParLog.ParList[CmdIndex] ;
	
	IF bWriteBusy OR bReadBusy THEN 
		bReady		:= FALSE;
		bBussy 		:= TRUE ;
		nProgress 	:= (100 / Param_Settings.MAX_PARAMETERS)* nRow ;
	ELSE
		bReady		:= TRUE	;
		bBussy 		:= FALSE;
		nProgress 	:= (100 / Param_Settings.MAX_PARAMETERS)* nRow ;
	END_IF

METHOD PRIVATE Mod_SearchIndex : BOOL
VAR_INPUT
END_VAR
// ====== set scroll index ======
	IF rtCmdScrollUp.Q THEN 
		 CmdIndex := CmdIndex + 1 ;
	ELSIF rtCmdScrollDown.Q THEN 
		 CmdIndex := CmdIndex - 1 ;
	END_IF 	 
	
// check if index number is within reach and if parameter is active
	IF CmdIndex > Param_Settings.MAX_PARAMETERS THEN 
		CmdIndex := 0 ;
	ELSIF CmdIndex < 0 THEN
		CmdIndex := Param_Settings.MAX_PARAMETERS ;
	END_IF

	IF NOT stParLog.ParList[CmdIndex].bActive AND bCmdScrollUp THEN // go to next index if parameter is not active 
		IF CmdIndex < Param_Settings.MAX_PARAMETERS THEN
			CmdIndex := CmdIndex + 1 ;
		ELSE
			CmdIndex := 0 ;
		END_IF
	ELSIF NOT stParLog.ParList[CmdIndex].bActive AND bCmdScrollDown THEN // go to previous index if parameter is not active 
		IF CmdIndex > 0 THEN
			CmdIndex := CmdIndex - 1 ;
		ELSE
			CmdIndex := Param_Settings.MAX_PARAMETERS ;
		END_IF
	ELSIF NOT stParLog.ParList[CmdIndex].bActive THEN
		IF CmdIndex < Param_Settings.MAX_PARAMETERS THEN
			CmdIndex := CmdIndex + 1 ;
		ELSE
			CmdIndex := 0 ;
		END_IF
	END_IF

// at new index set prep value to current value
	IF bCmdScrollUp OR bCmdScrollDown THEN 
		PrepValue := stParLog.ParList[CmdIndex].Value ;
	END_IF
END_METHOD

METHOD PUBLIC Mod_WriteTeachValue : BOOL
VAR_INPUT
		nCmdTeachPar	: UDINT	; // Name of parameter to be overwritten by teach value
		nCmdTeachValue	: LREAL	:= 0 		; // value from parameter teach
END_VAR
IF NOT bCmdTeach THEN 
	IF nCmdTeachPar <= Param_Settings.MAX_PARAMETERS AND nCmdTeachPar >= 0 THEN 
		CmdIndex 	:= nCmdTeachPar 	; 
		PrepValue 	:= nCmdTeachValue 	; 
		bCmdTeach	:= TRUE 			;
	END_IF
END_IF
END_METHOD

END_FUNCTION_BLOCK

// Parameter/Functions/Fb_ParLogging
FUNCTION_BLOCK PUBLIC Fb_ParLogging
VAR_OUTPUT
	stParLog		: Udt_ParLog ; // active parameter list
	bReadBusy		: BOOL		:= FALSE	; // File acces Bussy
	bWriteBusy		: BOOL 		:= FALSE	; // file write bussy
	bFryRead		: BOOL 		:= FALSE	; // File read done
	bFryWrite		: BOOL 		:= FALSE 	; // File Write Done 
	bError			: BOOL		:= FALSE	; // File acces error
	nErrId			: UDINT		:= 0		; // File acces error Id
	bValid 			: BOOL 		:= 0 		; // file write valid
	nRow	 		: UDINT 	:= 0		;(* Row number (record) *)
	nColumn			: UDINT 	:= 0	;(* Column number (record field) *)
END_VAR
VAR
	// ====== Internal commands ======
		bCmdWriteAllPar		: BOOL ;
		bCmdReadAllPar		: BOOL ; 
		StParameter			: UDT_Parameter_1 ;
		
	// ====== internal status ======
		bInitDone			: BOOL := FALSE ; // Init has been done  	
	// ====== Current step =====
		Step				: INT 	:= 0 	; // write action stepper
	
	// ====== Read variables ======
		hFile				: UINT	:= 0;(* File handle of the source file *)
		cbDone				: UDINT := 0;(* Counts allready parsed data bytes *)
		record				: ARRAY[0..1024] OF BYTE;(* Binary row data buffer. The size of this buffer have to be > length of longest record line + 2 (CRLF)  *)
		cbRecord			: UDINT := 0;(* Number of bytes in row buffer *)
		cbField				: UDINT	;(* Number of bytes in field buffer *)

	// ====== Write variables ======
		sParameterString	: ARRAY [0..Param_Settings.PAR_COLUMNS] OF STRING (Param_Settings.MAX_CSV_FIELD_LENGTH); (* temporary parameter buffer to string*)
		sCSVLine			: T_MaxString := '';(* Single CSV text line (row, record), we are using string as record buffer (your are able to see created fields) *)
		sCSVField			: T_MaxString := '';(* Single CSV field value (column, record field) *)
		
	// ====== Functions ======
		fbFileOpen		: FB_FileOpen	;(* Opens file *)
		fbFileClose		: FB_FileClose	;(* Closes file *)
		fbFileGets		: FB_FileGets	;(* Reads one record (line) *)
		fbFilePuts		: FB_FilePuts	;(* Writes one record (line) *)
		fbReader		: FB_CSVMemBufferReader;(* Helper function block used to parse CSV data bytes (single record line) *)
		fbWriter		: FB_CSVMemBufferWriter;(* Helper function block used to create CSV data bytes (single record line) *)
	
END_VAR

// ===== init =====
	IF NOT bInitDone THEN 
		Init();
	END_IF

// ===== Read parameters ====
	Mod_CSVFileRead();

// ====== Write parameter(s) to .csv ======
	Mod_CSVFileWrite();

METHOD PUBLIC Init : BOOL
VAR_INPUT
END_VAR
// Read parameters from .CSV file
	bCmdReadAllPar := TRUE ;

	IF bReadBusy THEN
		bInitDone := TRUE ;
	END_IF
END_METHOD

METHOD PRIVATE Mod_CSVFileRead : BOOL
VAR_INPUT
END_VAR
VAR
	i : UDINT ; // index number
END_VAR
// ===== Wait for command =====
	IF bReadBusy THEN 
		;
	ELSIF bCmdReadAllPar THEN
		;
	ELSE
		RETURN ;
	END_IF

// ===== prepare for file read =====
CASE step OF
	0:	(* Wait for rising edge at bRead variable *)
		bReadBusy		:= TRUE;
		bCmdReadAllPar 	:= FALSE ;
		bError			:= FALSE;
		nErrId			:= 0;
		hFile			:= 0;
		nRow			:= 1;
		nColumn			:= 0;
		cbRecord		:= 0;
		cbDone 			:= 0;
		step 			:= 1;

	1:	(* Open source file *)
		fbFileOpen(  bExecute := FALSE  );
		fbFileOpen( sNetId := Param_Settings.sNetId, sPathName := Param_Settings.sPARLIST_FILE, nMode := FOPEN_MODEREAD OR FOPEN_MODETEXT,(* Open file in text mode! *)
					ePath := PATH_GENERIC, bExecute := TRUE );
		step := 2;

	2:(* Wait until open not busy *)
		fbFileOpen( bExecute := FALSE, bError => bError, nErrID => nErrID, hFile => hFile );
		IF NOT fbFileOpen.bBusy THEN
			IF NOT fbFileOpen.bError THEN
				step := 3;
			ELSE(* Error: file not found? *)
				step := 100;
			END_IF
		END_IF

	3:	(* Read single line (record) *)
		fbFileGets( bExecute := FALSE );
		fbFileGets( sNetId := Param_Settings.sNetId, hFile := hFile, bExecute := TRUE );
		step := 4;

	4:(* Wait until read not busy *)
		fbFileGets( bExecute := FALSE, bError => bError, nErrID => nErrID, sLine => sCSVLine );
		IF NOT fbFileGets.bBusy THEN
			IF NOT fbFileGets.bError THEN
				IF fbFileGets.bEOF THEN
					step := 10;(* End of file reached => Close source file *)
				ELSE

					(* FB_FileGets returns text line without the CR (carriage return) character.
					We have to restore the CR character (replace the $L character with $R$L characters) *)
					IF RIGHT( sCSVLine, 1 ) = '$L' THEN
						sCSVLine := REPLACE( sCSVLine, '$R$L', 2, LEN( sCSVLine ) );
					END_IF

					step := 5;
				END_IF
			ELSE(* Error *)
				step := 100;
			END_IF
		END_IF

	5:(* Parse single line (record) *)
		fbReader.eCmd := eEnumCmd_First;(* Read first field value *)
		REPEAT
			fbReader( pBuffer := ADR( sCSVLine ), cbBuffer := SIZEOF( sCSVLine ), getValue => sCSVField );
			IF fbReader.bOk THEN
				fbReader.eCmd := eEnumCmd_Next;(* Read next field value *)
				IF ( nRow <= Param_Settings.MAX_PARAMETERS ) THEN
					IF ( nColumn <= Param_Settings.PAR_COLUMNS ) THEN

						CASE nColumn OF
								0: // Index number for array [UDINT]							
									i						:= STRING_TO_UDINT(CSVFIELD_TO_STRING( sCSVField, FALSE ));(* TODO: Save or use the field value in your application *) 
									stParLog.ParList[i].IndexNumber	:= i ; 	
									stParLog.ParList[i].bActive		:= TRUE ;						
								1: // Number [int]
									stParLog.ParList[i].Number 		:= STRING_TO_INT(CSVFIELD_TO_STRING( sCSVField, FALSE ));(* TODO: Save or use the field value in your application *)							
								2: // Name [String]
									stParLog.ParList[i].Name 		:= CSVFIELD_TO_STRING( sCSVField, FALSE );(* TODO: Save or use the field value in your application *)							
								3: // Par_Type E_paramterType [INT]
									stParLog.ParList[i].Par_Type	:= CSVFIELD_TO_STRING( sCSVField, FALSE );(* TODO: Save or use the field value in your application *)							
								4: // Discription [String]
									stParLog.ParList[i].Discription	:= CSVFIELD_TO_STRING( sCSVField, FALSE );(* TODO: Save or use the field value in your application *)							
								5: // Factory Value [LREAL]
									stParLog.ParList[i].Factory		:= STRING_TO_LREAL(CSVFIELD_TO_STRING( sCSVField, FALSE ));(* TODO: Save or use the field value in your application *)							
								6: // Maximum value [LREAL]
									stParLog.ParList[i].Maximum		:= STRING_TO_LREAL(CSVFIELD_TO_STRING( sCSVField, FALSE ));(* TODO: Save or use the field value in your application *)							
								7: // Minimum Value {LREAL]
									stParLog.ParList[i].Minimum 	:= STRING_TO_LREAL(CSVFIELD_TO_STRING( sCSVField, FALSE ));(* TODO: Save or use the field value in your application *)							
								8: // Unit	{String]
									stParLog.ParList[i].Unit		:= CSVFIELD_TO_STRING( sCSVField, FALSE );(* TODO: Save or use the field value in your application *)							
								9: // Value [LREAL]
									stParLog.ParList[i].Value 		:= STRING_TO_LREAL(CSVFIELD_TO_STRING( sCSVField, FALSE ));(* TODO: Save or use the field value in your application *)							
								10: // Saved {LREAL]	
									stParLog.ParList[i].Saved		:= STRING_TO_LREAL(CSVFIELD_TO_STRING( sCSVField, FALSE ));(* TODO: Save or use the field value in your application *)							
						ELSE
							;
						END_CASE
					END_IF
				END_IF
				nColumn := nColumn + 1;(* Increment number of read columns *)
				IF fbReader.bCRLF THEN(* CRLF == TRUE => End of reacord reached *)
					nRow 		:= nRow + 1;(* Increment number of read records *)
					nColumn 	:= 0;(* Reset number of columns *)
				END_IF
			ELSE(* Error: End of record reached or all fields read *)
				step := 3;(* Try to read next line *)
			END_IF
		UNTIL NOT fbReader.bOk
		END_REPEAT

	10:	(* Close source file *)
		fbFileClose( bExecute := FALSE );
		fbFileClose( sNetId := Param_Settings.sNetId, hFile := hFile, bExecute := TRUE );
		step := 11;

	11:(* Wait until close not busy *)
		fbFileClose( bExecute := FALSE, bError => bError, nErrID => nErrID );
		IF ( NOT fbFileClose.bBusy ) THEN
			hFile := 0;
			step := 100;
		END_IF

	100: (* Error or ready step => cleanup *)
		IF ( hFile <> 0 ) THEN
			step := 10; (* Close the source file *)
		ELSE
			bReadBusy := FALSE;
			step := 0;	(* Ready *)
		END_IF
END_CASE
END_METHOD

METHOD PRIVATE Mod_CSVFileWrite : BOOL
VAR_INPUT
END_VAR
// ===== Wait for command =====
	IF bWriteBusy THEN 
		;
	ELSIF bCmdWriteAllPar THEN 
		;
	ELSE
		RETURN ;
	END_IF

// ===== Start file write =====
CASE step OF
	0:	(* Wait for rising edge at bWrite variable *)
			bWriteBusy 			:= TRUE;
			bCmdWriteAllPar		:= FALSE ;
			bError				:= FALSE;
			nErrId				:= 0;
			hFile				:= 0;
			nRow				:= 0;
			nColumn				:= 0;
			step 				:= 1;
	1:	(* Open source file *)
		fbFileOpen(  bExecute := FALSE  );
		fbFileOpen( sNetId := Param_Settings.sNetId, sPathName := Param_Settings.sPARLIST_FILE, nMode := FOPEN_MODEWRITE OR FOPEN_MODETEXT,(* Open file in TEXT mode! *)
					ePath := PATH_GENERIC, bExecute := TRUE );
		step := 2;

	2:(* Wait until open not busy *)
		fbFileOpen( bExecute := FALSE, bError => bError, nErrID => nErrID, hFile => hFile );
		IF NOT fbFileOpen.bBusy THEN
			IF NOT fbFileOpen.bError THEN
				step := 3;
			ELSE(* Error: file not found? *)
				step := 100;
			END_IF
		END_IF

	3:(* Convert one PLC record to CSV format *)
		sCSVLine := '';
		fbWriter.eCmd := eEnumCmd_Next;(* Write first field value *)
		IF nRow <= Param_Settings.MAX_PARAMETERS THEN
			IF stParLog.ParList[nRow].bActive THEN // check if array row is active if not skip row (save proces time) 
				sParameterString[0] 	:= UDINT_TO_STRING (nRow);
				sParameterString[1] 	:= INT_TO_STRING(stParLog.ParList[nRow].Number);
				sParameterString[2] 	:= stParLog.ParList[nRow].Name;
				sParameterString[3] 	:= stParLog.ParList[nRow].Par_Type;
				sParameterString[4] 	:= stParLog.ParList[nRow].Discription;
				sParameterString[5] 	:= LREAL_TO_STRING(stParLog.ParList[nRow].Factory);
				sParameterString[6] 	:= LREAL_TO_STRING(stParLog.ParList[nRow].Maximum);
				sParameterString[7] 	:= LREAL_TO_STRING(stParLog.ParList[nRow].Minimum);
				sParameterString[8] 	:= stParLog.ParList[nRow].Unit;
				sParameterString[9] 	:= LREAL_TO_STRING(stParLog.ParList[nRow].Value);
				sParameterString[10]	:= LREAL_TO_STRING(stParLog.ParList[nRow].Saved);

				FOR nColumn := 0 TO Param_Settings.PAR_COLUMNS BY 1 DO
					sCSVField := STRING_TO_CSVFIELD( sParameterString[nColumn ], FALSE );(* TODO: Get field value from your application *)
	
					(* Add new field to the record buffer *)
					fbWriter( 	pBuffer := ADR( sCSVLine ), cbBuffer := SIZEOF( sCSVLine ) - 1, putValue := sCSVField, pValue := 0, cbValue := 0,
								bCRLF := ( nColumn = Param_Settings.PAR_COLUMNS ) );(* bCRLF == TRUE => Write CRLF after the last field value *)
					IF NOT fbWriter.bOk THEN
						step := 100;
						RETURN;
					END_IF
				END_FOR(* FOR nColumn := 0... *)
	
				(* FB_FilePuts adds allready CR (carriage return) to the written line.
				We have to replace the $R$L characters with $L character to avoid double CR. *)
				IF RIGHT( sCSVLine, 2 ) = '$R$L' THEN
					sCSVLine := REPLACE( sCSVLine, '$L', 2, LEN( sCSVLine ) - 1 );
				END_IF
	
				nRow := nRow + 1;(* Increment number of created records (rows) *)
				step := 4;(* Write record to the file *)
			ELSE 
				nRow := nRow +1 ;(* Increment number of created records (rows) *)
			END_IF							
		ELSE(* All rows written => Close file *)
			step := 10;
		END_IF

	4:	(* Write single text line *)
		fbFilePuts( bExecute := FALSE );
		fbFilePuts( sNetId := Param_Settings.sNetId, hFile := hFile, sLine := sCSVLine, bExecute := TRUE );
		step := 5;

	5:(* Wait until write not busy *)
		fbFilePuts( bExecute := FALSE, bError => bError, nErrID => nErrID );
		IF NOT fbFilePuts.bBusy THEN
			IF NOT fbFilePuts.bError THEN
				step := 3;(* Write next record *)
			ELSE(* Error *)
				step := 100;
			END_IF
		END_IF

	10:	(* Close source file *)
		fbFileClose( bExecute := FALSE );
		fbFileClose( sNetId := Param_Settings.sNetId, hFile := hFile, bExecute := TRUE );
		step := 11;

	11:(* Wait until close not busy *)
		fbFileClose( bExecute := FALSE, bError => bError, nErrID => nErrID );
		IF ( NOT fbFileClose.bBusy ) THEN
			hFile := 0;
			step := 100;
		END_IF

	100: (* Error or ready step => cleanup *)
		IF ( hFile <> 0 ) THEN
			step := 10; (* Close the source file *)
		ELSE
			bWriteBusy := FALSE;
			step := 0;	(* Ready *)
		END_IF

END_CASE
END_METHOD

METHOD PUBLIC Mod_BackupPar : BOOL
VAR_INPUT
END_VAR
// ====== Set parameter write command ======
	IF NOT bWriteBusy AND NOT bReadBusy AND NOT bError THEN 
		bCmdWriteAllPar 	:= TRUE 	;
		Mod_BackupPar 		:= FALSE 	;	
	ELSE 
		Mod_BackupPar 	:= TRUE 	;	
	END_IF
END_METHOD

METHOD Mod_ChangePar : BOOL
VAR_INPUT
	stInputParameter 	: Udt_Parameter_2 ; // input parameter to be changed	
	i					: UDINT			; // index number of parameter
END_VAR
// write parameter to log
	IF NOT bWriteBusy AND NOT bReadBusy THEN 
		i 			:= stInputParameter.IndexNumber ; // check index number
		IF i <= Param_Settings.MAX_PARAMETERS THEN
			stParLog.ParList[i] 	:= stInputParameter ;
		END_IF
	END_IF
END_METHOD

METHOD PUBLIC Mod_ReadAllPar : BOOL
VAR_INPUT
END_VAR
// ====== Set parameter Read command ======
	IF NOT bWriteBusy AND NOT bReadBusy AND NOT bError THEN 
		bCmdReadAllPar 		:= TRUE ;
		Mod_ReadAllPar 		:= FALSE;	
	ELSE 
		Mod_ReadAllPar 		:= TRUE ;	
	END_IF
END_METHOD

END_FUNCTION_BLOCK

// PathFunctions/F_FBNameFromPath
FUNCTION F_FBNameFromPath : STRING // distills .fb name from function path
VAR_INPUT
	sPath	: STRING ;
END_VAR
VAR
	sTemp		: STRING ;
	nstartFbName: INT ; 
END_VAR

sTemp := sPath ;

REPEAT 
	// Look for first occurance of .fb in string
	nStartFbName := FIND( sTemp,'.fb');
	// Delete text before .fb and .fb itself
	IF nstartFbName <>0 THEN 
		sTemp := DELETE( STR := sTemp, LEN := nstartFbName + 3, 0); 
	END_IF
UNTIL
	nstartFbName = 0 
END_REPEAT

F_FBNameFromPath := sTemp ;

END_FUNCTION

// Positions/FunctionBlocks/FB_PositionTrigger
FUNCTION_BLOCK PUBLIC FB_PositionTrigger // trigger function, sets trigger Q signal high when trigger position is between previous cycle's and current axis position.
VAR_INPUT
	fAxisPos			: LREAL	; // Axis position on which the to trigger
	nAxisModuloRev		: DINT 	:= 0	; // axis modulo revolutions 
	fAxisVelocity		: LREAL := 0 	; 	// velocity of axis 
	bDirPositive		: BOOL 	:= TRUE ; // Axis direction is forward 
	fEncoderTurnover	: LREAL	:= 360 	; // Encoder turnover value (standard 360 deg)
	bEnablenNegative 	: BOOL 	:= FALSE; // Enables negative input values
END_VAR
VAR_OUTPUT
	Q					: BOOL 	; // trigger signal
	bInternalTrigger	: BOOL 	; // Internal trigger signal 
	bTriggerArmed 		: BOOL 	; // Trigger is armed 
	bEncoderTurnedOver	: BOOL 	; // is high when encoder goes thru it's turnover point 
	fAccuracy 			: LREAL ; // Accuracy of trigger 
END_VAR
VAR
	// function commands
	fTriggerPosition 		: LREAL ; // trigger position 
	fTriggerPosCompensated	: LREAL ; // TRigger Position after compensation
	nRotBeforeTrigger		: DINT 	:= 0 ; 	// Full axis rotations before position trigger is armed
	nRotBeforeTriggerCompensated	: DINT := 0 ; // full E_ComponentTypes.Axis rotation before trigger IsFinite armed 
	// Trigger variables 
	fReactionTime			: LREAL	:= 0 ; 	// [ms] Time before reaction to trigger (time compensation)
	// internal values	
	nTriggerRotation		: DINT	:= 0 ; 	// Number of rotations done since trigger is armed 
	fOldAxisPos				: LREAL ; 		// Old axis position for comparison
	nOldAxisRev				: DINT 	; 		// Old modulo revolutions 
	fCompensationDistance	: LREAL := 0 ; 	// [units] trigger compensation distance  
	// Edge functions 
	fbReTriggerArmed		: R_TRIG ; // rising edge trigger on trigger armed (used to rest trigger values) 
END_VAR

// Rising edge function execute
fbReTriggerArmed(CLK := bTriggerArmed); 

// ==== Skip function if trigger is not armed =====
	IF NOT bTriggerArmed THEN  
		bInternalTrigger	:= FALSE 	;
		RETURN ;	
	ELSIF fbReTriggerArmed.Q THEN 
		fOldAxisPos 		:= fAxisPos ;
		nOldAxisRev			:= nAxisModuloRev ;
		nTriggerRotation	:= 0 		; 
		Q 					:= FALSE	;
	END_IF

// ==== check if encoder is at turnover =====
	ExecTurnoverCheck(); 
// ==== compare positions to trigger ======
	CalcTriggerCompensation();
	ExecArmTrigger();

METHOD PRIVATE CalcTriggerCompensation : BOOL
VAR_INPUT
END_VAR
// ===== Calculate the distance travelled within the delay time =====
	fCompensationDistance	:= fReactionTime  * (fAxisVelocity / 1000);
END_METHOD

METHOD INTERNAL ExecArmTrigger : BOOL
VAR_INPUT
END_VAR
// ===== Retract compensationdistance from trigger distance =====

// check if trigger pos is not negative 
IF NOT bEnablenNegative AND fTriggerPosCompensated < 0 THEN
	fTriggerPosCompensated 			:= fEncoderTurnover + fTriggerPosition ;
	nRotBeforeTriggerCompensated	:= nRotBeforeTrigger -	1;  
ELSE
	fTriggerPosCompensated 			:= fTriggerPosition - fCompensationDistance ;
	nRotBeforeTriggerCompensated	:= nRotBeforeTrigger ;  
END_IF 

// ==== compare positions to trigger ======
	bInternalTrigger := FALSE ;

	IF bEncoderTurnedOver THEN
		IF bDirPositive THEN
			bInternalTrigger S= Between(fOldAxisPos , fTriggerPosCompensated, fEncoderTurnover) ;
			bInternalTrigger S= Between(0	, fTriggerPosCompensated, fAxisPos) ;
		ELSE 
			bInternalTrigger S= Between(0			, fTriggerPosCompensated, fOldAxisPos) ;
			bInternalTrigger S= Between(fAxisPos	, fTriggerPosCompensated, fEncoderTurnover) ;
		END_IF 
		bEncoderTurnedOver := FALSE ;
	ELSE 
		bInternalTrigger S= Between(fAxisPos	, fTriggerPosCompensated, fOldAxisPos) ;
		bInternalTrigger S= Between(fOldAxisPos	, fTriggerPosCompensated, fAxisPos) ;
		fAccuracy	:= ABS( fOldAxisPos - fAxisPos);
	END_IF

	fOldAxisPos := fAxisPos ;

// ==== Check multiturn command =======
	IF bInternalTrigger THEN 
		IF nTriggerRotation >= nRotBeforeTriggerCompensated THEN 
			Q S= bInternalTrigger;			
		ELSE 
			nTriggerRotation := nTriggerRotation + 1 ;
		END_IF 
	END_IF

// ==== Reset arm trigger command =====
	bTriggerArmed R= Q ;
END_METHOD

METHOD PRIVATE ExecTurnoverCheck : BOOL
VAR_INPUT
END_VAR
	bEncoderTurnedOver := nOldAxisRev <> nAxisModuloRev ;
	nOldAxisRev := nAxisModuloRev ;
END_METHOD

METHOD PUBLIC CmdArmTrigger : BOOL // arm trigger
VAR_INPUT
END_VAR
// Arm trigger command 
bTriggerArmed S= TRUE ;

// set feedback
CmdArmTrigger := NOT Q ;
END_METHOD

METHOD PUBLIC CmdSetTriggerPos : BOOL
VAR_INPUT
	fCmdPosition 	: LREAL ; // Trigger position 
	nCmdRotations	: DINT	:= 0 ; // Rotations before trigger is set  
	nCmdReactionTime: LREAL := 0 ; // [ms]reaction time to trigger signal 
END_VAR
// set trigger position
fTriggerPosition 	:= fCmdPosition ;
nRotBeforeTrigger	:= nCmdRotations;
fReactionTime 		:= nCmdReactionTime ;
END_METHOD

END_FUNCTION_BLOCK

// Positions/Functions/F_AccDecDistanceFromTime
FUNCTION F_AccDecDistanceFromTime : LREAL
VAR_INPUT
	nAccelDecel	: LREAL ; // acceleration or deceleration [units/s^2]
	nTimeMs		: LREAL	; // Time for acceleratio/ deceleration to take place [ms]
END_VAR
VAR
	nTimeSec	: LREAL;
	nVelocity	: LREAL;
END_VAR

nTimeSec := nTimeMs/1000;

nVelocity := nAccelDecel * nTimeSec;

F_AccDecDistanceFromTime := nVelocity * nTimeSec / 2 ;

END_FUNCTION

// Positions/Functions/F_AccDecDistanceFromVelo
FUNCTION F_AccDecDistanceFromVelo : LREAL
VAR_INPUT
	nVelocity	: LREAL ; // velocity [m/s]
	nAccDecc	: LREAL ; // acceleration or deceleration value [m/s^2]
END_VAR
VAR
	nTime : LREAL ;
END_VAR

nTime := nVelocity	/	nAccDecc ;

F_AccDecDistanceFromVelo := nVelocity * (nTime/2);

END_FUNCTION

// Positions/Functions/F_PosCheck
(* Returns a true when position is within tollerance *)
FUNCTION F_PosCheck : bool
VAR_INPUT
	TargetPos		: LREAL ; // target position to check [deg]
	ActPos			: LREAL	; // Actual position [deg]
	Lowtol			: LREAL	; // Low tolerance (is reduced from target pos)
	HighTol			: LREAL	; // High tollerance (is added to target position)
	EncTurnover		: DINT 	; // Encoder turnover value
END_VAR
VAR
	Lowval	: LREAL ;
	HighVal	: LREAL ;
	LowTurn	: BOOL ;
	HighTurn: BOOL ;
	HighOk	: BOOL ;
	LowOK	: BOOL ;
END_VAR

// Check lower and uper do not exceed turnover
	IF TargetPos - Lowtol < 0 THEN 
		Lowval 	:= EncTurnover + TargetPos - Lowtol ;
		LowTurn	:= TRUE ;
	ELSE 
		LowTurn := FALSE ;
	END_IF

	IF TargetPos + HighTol > 360 THEN 
		HighVal	:= EncTurnover - TargetPos + Lowtol ;
		HighTurn:= TRUE ;
	ELSE 
		HighTurn := FALSE ;
	END_IF

	
// Check lower limit
	IF ActPos > TargetPos - Lowtol THEN
		LowOK := TRUE ;
	ELSIF LowTurn AND ActPos > Lowval THEN
		LowOK := TRUE ; 
	ELSIF HighTurn AND ActPos < HighVal THEN 
		LowOK := TRUE ;
	ELSE 
		LowOK := FALSE ;
	END_IF
	
// Check high limit
	IF ActPos < TargetPos + HighTol THEN
		HighOk := TRUE ;
	ELSIF HighTurn AND ActPos < HighVal THEN
		HighOk := TRUE ;
	ELSIF LowTurn AND ActPos > Lowval THEN 
		HighOk := TRUE ; 
	ELSE
		HighOk := FALSE ;
	END_IF
	
// Set output
	IF LowOK AND HighOk THEN
		F_PosCheck := TRUE ;
	ELSE 
		F_PosCheck := FALSE ;
	END_IF

END_FUNCTION

// Positions/Functions/F_TopVelocityFromTime
FUNCTION F_TopVelocityFromTime : LREAL
VAR_INPUT
	nAccel	: LREAL ; // acceleration or deceleration [units/s^2]
	nTimeMs		: LREAL	; // Time for acceleratio/ deceleration to take place [ms]
END_VAR
VAR
	nTimeSec	: LREAL;
END_VAR

nTimeSec := nTimeMs/1000;

F_TopVelocityFromTime := nAccel * nTimeSec;

END_FUNCTION

// Positions/Functions/F_TriggerPosOffset
(* function to calculate trigger points for time based moves *)
FUNCTION F_TriggerPosOffset : LREAL
VAR_INPUT
	Velocity		: LREAL	; // [Units/sec] command velocity 
	nMoveTimeMs		: LREAL	; // [ms] Time it takes for move to complete
END_VAR
VAR
END_VAR

// ===== Convert time to usable calculation value =====
	F_TriggerPosOffset := nMovetimeMs * ABS(Velocity / 1000);

END_FUNCTION

// System/Functions/DataManagement/FB_PersistentDataManager
FUNCTION_BLOCK FB_PersistentDataManager
VAR_INPUT
END_VAR
VAR_OUTPUT
END_VAR
VAR
	FbWritePersistentData : FB_WritePersistentData ;
	cmdWrite : BOOL := FALSE ;
	TOfWriteInterval	: TOf ;
	CmdWriteFromTime	: BOOL ; 
	TestjeWritten		: BOOL ;
END_VAR

// ===== persistent write interval =====
 TOfWriteInterval(	IN := cmdWrite OR NOT TOfWriteInterval.Q,
	 				PT	:= T#5M  );

IF NOT TOfWriteInterval.Q THEN 
	cmdWrite := TRUE ;
END_IF

// ===== write persistent data =====
	FbWritePersistentData ( PORT 	:= 851,
							START 	:= CmdWrite,
							TMOUT 	:= T#1S,	
							mode 	:= E_PersistentMode.SPDM_VAR_BOOST );	

IF cmdWrite AND FbWritePersistentData.BUSY THEN 
	cmdWrite := FALSE ;
END_IF

METHOD PUBLIC Write : BOOL
VAR_INPUT
END_VAR
IF NOT FbWritePersistentData.BUSY THEN 
	cmdWrite := TRUE ;
ELSE 
	Write := TRUE ;
END_IF
END_METHOD

END_FUNCTION_BLOCK

// System/Functions/Fb_SystemVariables
FUNCTION_BLOCK Fb_SystemVariables
VAR
	// **** Function blocks *****
		Fb_SystemTime: FB_LocalSystemTime ;
		Fb_TimerHbOn : Ton ; // Timer Heartbeat on
		Fb_TimerFast : Ton ; // Timer for fast blink bit
		Fb_TimerSlow : Ton ; // Timer for slow blink bit
		Fb_RisingPulse : R_Trig ; // Rinsing edge trigger function	

	// ***** internal Variables *****
		TimeStruct	: TIMESTRUCT ; // Time structure from system time function
		HeartbeatOn	: BOOL ; // heartbeat is on
		FlashFastOn	: BOOL ; // Fast Flash bit on
		FlashSlowOn	: BOOL ; // Flash slow bit on
		
END_VAR

// ===== Get system time =====
	// ***** get windows system time *****
		Fb_SystemTime(	sNetID := '', 
						bEnable := TRUE, 
						dwCycle := 1,
						dwOpt := 0, 
						tTimeout := DEFAULT_ADS_TIMEOUT, 	
						systemTime => TimeStruct,
						tzID	=> Sys_Variables.TimeZoneId
						);
	// ****** convert to time of day format *****
		Sys_Variables.SystemTime := SYSTEMTIME_TO_DT(TIMESTR := TimeStruct) ;

// ===== Heartbeat generator =====
	Fb_TimerHbOn(In := NOT HeartbeatOn , PT:= T#1S, Q => HeartbeatOn);
	IF Fb_TimerHbOn.ET >= T#500MS THEN
		Sys_Variables.HeartBeat := TRUE ;
	ELSE
		Sys_Variables.HeartBeat := FALSE ;
	END_IF

// ===== one second pulse generator =====
	Fb_RisingPulse(Clk := HeartbeatOn, Q => Sys_Variables.Pulse1Sec);

// ===== Flash fast bit =====
	Fb_TimerFast(In := NOT FlashFastOn, Pt := T#1S, Q => FlashFastOn);
	IF Fb_TimerFast.ET >= T#600MS THEN
		Sys_Variables.BlinkFast := TRUE;  
	ELSE
		Sys_Variables.BlinkFast := FALSE;  		
	END_IF
// ===== Flash Slow bit =====
	Fb_TimerSlow(In := NOT FlashSLowOn, Pt := T#2S, Q => FlashSlowOn);
	IF Fb_TimerSlow.ET >= T#1200MS THEN
		Sys_Variables.BlinkSlow := TRUE;  
	ELSE
		Sys_Variables.BlinkSlow := FALSE;  		
	END_IF

// ===== Always true and always false bits =====
	Sys_Variables.AlwaysOff := FALSE 	;
	Sys_Variables.AlwaysOn	:= TRUE		;
	
// ===== Manage persistent data ======
	DataManager.FbPersistentManager();

END_FUNCTION_BLOCK
